Fanuc KAREL source: kf00068.KL

-- PROVISIONAL review KL for V1013-1; original PC SHA256 0b908687eb816916cabb1e0c969ee605a50984b15a70656babf1f19052506e52
-- Incomplete behavior may be omitted. Consult companion uncertainty JSON. Do not deploy.
PROGRAM KF00068
%NOLOCKGROUP
VAR
  I : INTEGER
  J : INTEGER
  X : REAL
  Y : REAL
  B : BOOLEAN
  C : BOOLEAN
  TXT : STRING[80]
  TXT2 : STRING[80]
  STATUS : INTEGER
-- UNRESOLVED_DECL AI type=002010
-- UNRESOLVED_DECL BI type=002010
-- UNRESOLVED_DECL P type=000102
-- UNRESOLVED_DECL JP type=000199
-- UNRESOLVED_DECL PF type=000101
-- UNRESOLVED_DECL V1 type=000013
-- UNRESOLVED_DECL V2 type=000013
BEGIN
  -- UNRESOLVED_PC offsets 5-16; opcodes 2E,23
  -- UNRESOLVED_PC offsets 21-32; opcodes 2E,23
  -- UNRESOLVED_PC offsets 37-48; opcodes 2E,23
  -- UNRESOLVED_PC offsets 53-68; opcodes 27,22,76,23
  -- UNRESOLVED_PC offsets 73-77; opcodes 7F
END KF00068
